TYPE ST_CAMERA_Ctrl :    //ST_SCANNER_CameraMap
STRUCT
	bProcessNewCode		: BOOL;
	bManualTrigger		: BOOL;
	bConfigMode			: BOOL;	
	bResetStats			: BOOL;	
	
	stBrowseCtrl		: ST_CAMERA_BrowseCtrl;
	stCameraMap			: ST_CAMERA_Mapping;
END_STRUCT
END_TYPE

(* stored: Version 1.1.0.1
   DUT ST_CAMERA_Ctrl: Id {d8b1c7c7-f13e-4669-b41a-f9eda99bb635} *)
